// TIA Portal V17 export
// export: Created 2024-09-15T12:30:18.9225043Z, ExportSetting WithDefaults, DisplayName Totally Integrated Automation Portal, DisplayVersion V17, DisplayName TIA Portal Openness, DisplayVersion V17, DisplayName TIA Portal Version Control Interface, DisplayVersion V17, DisplayName STEP 7 Professional, DisplayVersion V17, DisplayName STEP 7 Safety, DisplayVersion V17, DisplayName WinCC Professional, DisplayVersion V17
VAR_GLOBAL   // PLC tag table "HBW - Automated High-Bay Warehouse"
   IX_HBW_RefSwitchHorizontalAxis_I1 AT %I1.0 : Bool;   // HBW - I1 = Reference switch horizontal axis   {ExternalAccessible false, ExternalVisible false, ExternalWritable false}
   IX_HBW_LightBarrierInside_I2 AT %I1.1 : Bool;   // HBW - I2 = Light barrier inside   {ExternalAccessible false, ExternalVisible false, ExternalWritable false}
   IX_HBW_LightBarrierOutside_I3 AT %I1.2 : Bool;   // HBW - I3 = Light barrier outside   {ExternalAccessible false, ExternalVisible false, ExternalWritable false}
   IX_HBW_RefSwitchVerticalAxis_I4 AT %I1.3 : Bool;   // HBW - I4 = Reference switch vertical axis   {ExternalAccessible false, ExternalVisible false, ExternalWritable false}
   IX_HBW_TrailSensor1Lower_A1 AT %I5.0 : Bool;   // HBW - A1 = Trail sensor (signal 1, lower)   {ExternalAccessible false, ExternalVisible false, ExternalWritable false}
   IX_HBW_TrailSensor2Upper_A2 AT %I5.4 : Bool;   // HBW - A2 = Trail sensor (signal 2, upper)   {ExternalAccessible false, ExternalVisible false, ExternalWritable false}
   IX_HBW_EncoderVerticalAxisImp1_B3 AT %I5.2 : Bool;   // HBW - B3 = Encoder vertical axis imulse 1   {ExternalAccessible false, ExternalVisible false, ExternalWritable false}
   IX_HBW_EncoderVerticalAxisImp2_B4 AT %I5.6 : Bool;   // HBW - B4 = Encoder vertical axis imulse 2   {ExternalAccessible false, ExternalVisible false, ExternalWritable false}
   IX_HBW_EncoderHorizontalAxisImp1_B1 AT %I5.1 : Bool;   // HBW - B1 = Encoder horizontal axis imulse 1   {ExternalAccessible false, ExternalVisible false, ExternalWritable false}
   IX_HBW_EncoderHorizontalAxisImp2_B2 AT %I5.5 : Bool;   // HBW - B2 = Encoder horizontal axis imulse 2   {ExternalAccessible false, ExternalVisible false, ExternalWritable false}
   IX_HBW_SwitchCantileverFront_I5 AT %I1.4 : Bool;   // HBW - I5 = Reference switch cantilever front   {ExternalAccessible false, ExternalVisible false, ExternalWritable false}
   IX_HBW_SwitchCantileverBack_I6 AT %I1.5 : Bool;   // HBW - I6 = Reference switch cantilever back   {ExternalAccessible false, ExternalVisible false, ExternalWritable false}
   QX_HBW_M1_ConveyorBeltForward_Q1 AT %Q1.0 : Bool;   // HBW - Q1 = Motor M1 conveyor belt forward   {ExternalAccessible false, ExternalVisible false, ExternalWritable false}
   QX_HBW_M1_ConveyorBeltBackward_Q2 AT %Q1.1 : Bool;   // HBW - Q2 = Motor M1 conveyor belt backward   {ExternalAccessible false, ExternalVisible false, ExternalWritable false}
   QX_HBW_M2_HorizontalTowardsRack_Q3 AT %Q1.2 : Bool;   // HBW - Q3 = Motor M2 horizontal towards rack   {ExternalAccessible false, ExternalVisible false, ExternalWritable false}
   QX_HBW_M2_HorizontalTowardsConveyorBelt_Q4 AT %Q1.3 : Bool;   // HBW - Q4 = Motor M2 horizontal towards conveyor belt   {ExternalAccessible false, ExternalVisible false, ExternalWritable false}
   QX_HBW_M3_VerticalAxisDownward_Q5 AT %Q1.4 : Bool;   // HBW - Q5 = Motor M3 vertical axis downward   {ExternalAccessible false, ExternalVisible false, ExternalWritable false}
   QX_HBW_M3_VerticalAxisUpward_Q6 AT %Q1.5 : Bool;   // HBW - Q6 = Motor M3 vertical axis upward   {ExternalAccessible false, ExternalVisible false, ExternalWritable false}
   QX_HBW_M4_CantileverForward_Q7 AT %Q1.6 : Bool;   // HBW - Q7 = Motor M4 cantilever forward   {ExternalAccessible false, ExternalVisible false, ExternalWritable false}
   QX_HBW_M4_CantileverBackward_Q8 AT %Q1.7 : Bool;   // HBW - Q8 = Motor M4 cantilever backward   {ExternalAccessible false, ExternalVisible false, ExternalWritable false}
   QW_HBW_PWM_ConveyorBelt_M1 AT %QW7 : Int;   // HBW = PWM Motor M1 conveyor belt   {ExternalAccessible false, ExternalVisible false, ExternalWritable false}
   QW_HBW_PWM_HorizontalAxis_M2 AT %QW9 : Int;   // HBW = PWM Motor M2 horizontal axis   {ExternalAccessible false, ExternalVisible false, ExternalWritable false}
   QW_HBW_PWM_VerticalAxis_M3 AT %QW11 : Int;   // HBW = PWM Motor M3 vertical axis   {ExternalAccessible false, ExternalVisible false, ExternalWritable false}
   QW_HBW_PWM_Cantilever_M4 AT %QW13 : Int;   // HBW = PWM Motor M4 cantilever   {ExternalAccessible false, ExternalVisible false, ExternalWritable false}
END_VAR
